// Mitsubishi GX Works2 project: vent_v02   PLC: FX3G
// Базовая структура управления вентиляциооной установкой

// global labels: Global1
VAR_GLOBAL
  xStart AT M10 : BOOL;  (* Переменная разрешения на работу установки *)
  xSeason AT M12 : BOOL;  (* Определение сезона 0 - Зима 1 - Лето *)
  xAlarm AT M1 : BOOL;  (* Общий статус Аварий 0 - нет 1 - Авария *)
  xWarning AT M2 : BOOL;  (* Общий статус предупреждений 0 - нет 1 - есть предупреждения *)
  dI_AlarmFreeze AT X000 : BOOL;  (* Авария термостата заморозки *)
  xAlarmSensors AT M7 : BOOL;  (* Общая аврия Датчиков - всне диапазона *)
  dI_AlarmPumpWater AT X001 : BOOL;  (* Авария насоса (сработка защиты) *)
  dI_AlarmMotorSupply AT X002 : BOOL;  (* Авария реле Вентилятора Притока *)
  dI_AlarmMotorExhaust AT X003 : BOOL;  (* Авария реле Вентилятора Вытяжки *)
  dI_WarnPresFilterSupply AT X007 : BOOL;  (* Авария пресостата фильтра Притока *)
  dI_WarnPresFilterExaust AT X006 : BOOL;  (* Авария пресостата фильтра Вытяжки *)
  dI_AlarmPresMotorSupply AT X004 : BOOL;  (* Авария пресостата вентилятора Притока *)
  dI_AlarmPresMotorExhaust AT X005 : BOOL;  (* Авария пресостата вентилятора Вытяжки *)
  xAlarmWarmWater AT M8 : BOOL;  (* Авария снижения температуры теплоносителя темплообменника - Требуется прогрев *)
  wDeltaTempOut AT D11 : INT;  (* Значение смещения показаний датчика (корректировка) *)
  wDeltaTempInRoom AT D10 : INT;  (* Значение смещения показаний датчика (корректировка) *)
  wDeltaTempFromRoom AT D9 : INT;  (* Значение смещения показаний датчика (корректировка) *)
  wDeltaTempEmpty AT D8 : INT;  (* Значение смещения показаний датчика (корректировка) *)
  xAlarmSensorOut AT M6 : BOOL;  (* Авария датчика Наружней температуры *)
  xAlarmSensorInRoom AT M5 : BOOL;  (* Авария датчика температуры Подачи В помещение *)
  xAlarmSensorFromRoom AT M4 : BOOL;  (* Авария датчика температуры забираемого ИЗ помещения *)
  xAlarmSensorEmpty AT M3 : BOOL;  (* Авария датчика температуры *)
  iR_TempOut AT D6 : WORD;  (* Значение сопротивление линии связи резистивного датчика *)
  iR_TempInRoom AT D5 : WORD;  (* Значение сопротивление линии связи резистивного датчика *)
  iR_TempFromRoom AT D4 : WORD;  (* Значение сопротивление линии связи резистивного датчика *)
  iRTempEmpty AT D7 : WORD;  (* Значение сопротивление линии связи резистивного датчика *)
  dO_PumpStart AT Y004 : BOOL;  (* Разрешение на работу Насоса контура водяного теплообменника *)
  dO_SupplyMotorStart AT Y003 : BOOL;  (* Разрешение на запуск Вентилятора Притока *)
  dO_ExhaustMotorStart AT Y001 : BOOL;  (* Разрешение на запуск Вентилятора Вытяжки *)
  dO_SupplyDamperStart AT Y002 : BOOL;  (* Разрешение на открытие Заслонки Притока *)
  dO_ExhaustDamperStart AT Y000 : BOOL;  (* Разрешение на открытие Заслонки Вытяжки *)
  iDelayStart AT D131 : WORD;  (* Значение задержки (общее) *)
  iDelaySupplyMotor AT D3 : WORD;  (* Значение задержки пуска Вентилятора Притока *)
  iDelayExhaustMotor AT D1 : WORD;  (* Значение задержки пуска Вентилятора Вытяжки *)
  iDelayDamper AT D132 : WORD;  (* Значение задержки открытия заслонки *)
  xUserStart AT M11 : BOOL;  (* Переменная изменяемая Пользователем для разрешения работы *)
  xUserSeason AT M13 : BOOL;  (* Переменная изменяемая Пользователем для выбора Сезона *)
  xUserArarmReset AT M14 : BOOL;  (* Переменная изменяемая Пользователем для сброса общего флага Аварий *)
  xAlarmCritical AT M0 : BOOL;  (* Cтатус критических Аварий 0 - нет 1 - Авария *)
  xInit AT M15 : BOOL;  (* Переменная разрешающая иницилизацию при старте *)
  aI_TempOut AT D14 : INT;  (* AI_0 Датчик наружней температуры D8030 *)
  aI_TempSupply AT D15 : INT;  (* AI_1 Датчик притока (температуры подачи в помещение)  D8031 *)
  aI_TempWater AT D16 : INT;  (* AI_2 Датчик обратной воды  D8032 *)
  aI_TempRecupOut AT D17 : INT;  (* AI_3 Датчик температуры за рекуператором  D8033 *)
  aO_1 AT D8050 : REAL;  (* AO_ Первый аналоговый D8050 *)
  aO_2 AT D8051 : REAL;  (* AO_ Второй аналоговый выход D8051 *)
  iUserTempSummer AT D128 : INT;  (* Температура перехода на летний режим *)
  iUserTemWinter AT D129 : INT;  (* Температура перехода на зимний режим *)
  aI_TempFromRoom AT D18 : INT;  (* AI_4 Датчик вытяжной температуры из помещения D8034 *)
  iUserAccess AT D40 : WORD;  (* Уровень доступа текущего пользователя *)
  iUserSetpointTempSupply AT D130 : INT;  (* Уставка заданная пользователем *)
  testTempOut AT D41 : INT;  (* Тестирование перехода   Зима/Лето *)
  iSetpointTempSupply AT D20 : INT;  (* Уставка температуры подачи Системная *)
  iUserSetpointTempWater AT D133 : INT;  (* Уставка контроля температуры теплоносителя (вода) *)
  iUserSetpointTempGlycol AT D134 : INT;  (* Уставка контроля температуры теплоносителя гликоль *)
  iUserSetpointTempAlarm AT D135 : INT;  (* Уставка контроля температуры Аварии *)
END_VAR

// task Task_01 (event TRUE, interval 0, priority 31): POU_01
// task Init (event M8002, interval 0, priority 24): Init
// task Process (event FALSE, interval T#150ms, priority 29): Process
// user libraries (not included): AlarmManger128v11, Utils

PROGRAM Init
VAR
  fbAmSet : AM_SET;
  fbAmInit : AM_INIT;
  fbAmIs : AM_HAS_ALARMS;
  fbAmBlockIs : AM_IS_BLOCK;
  fbAmEvents : AM_EVENT;
  fbAmRST : AM_RST;
  fbAmEventRST : AM_EVENT_RESET;
  inputType : BOOL;
END_VAR
(*Programm is run only one time when plc started to initiate alarms,  warnings and configuration settings *)


	AM_D_START :=3000; (* Start alarms library*)
	
	(* Critical Alarm signals*)
	 fbAmInit(iNum := 0, iSeverity :=3, iProcess :=1, xLock := TRUE,  xLatch := TRUE,  xBuzzer := TRUE ); (*Fire alarm *) 
	 
	  fbAmInit(iNum := 1, iSeverity :=2, iProcess :=2, xLock := TRUE,  xLatch := FALSE,  xBuzzer := TRUE ); (*Sensor alarm *) 


(* *)
END_PROGRAM

PROGRAM POU_01
VAR
  iStep : INT;
  fbAmSet : AM_SET;
  fbAmInit : AM_INIT;
  fbAmIs : AM_HAS_ALARMS;
  fbAmBlockIs : AM_IS_BLOCK;
  fbAmEvents : AM_EVENT;
  fbAmRST : AM_RST;
  fbAmEventRST : AM_EVENT_RESET;
  localSeasonTriger : BOOL;
  icountMin : INT;
  init : INT;
  currentTemp : INT;
  couner : INT;
END_VAR
(* RST( MEP( xManualWorks ) , xAutoWorks );
RST( MEP(xAutoWorks ) ,xManualWorks  );  *)
(* System can work only in one state Auto or Manual There is constol change*)
	
		fbAmIs(iProcessNum:= 2 ,iSeverity:= 2 ,Q:= xAlarmSensors);
		fbAmIs(iProcessNum:= 1, iSeverity:= 3 ,Q:= xAlarm );
 		IF xInit = 0 OR xAlarm THEN  iStep := 0 ; 
 		ELSE 
 			iStep := 10;
 		END_IF; (* Проверяем была ли выполнена инициализация xInit = 1 Ули была то переходим на шаг 10 если нет - на шаг 0 *)

fbAmRST(IN:= M10 );

CASE iStep OF
	0: (* Init  - Инициализация Задаем начальные значения переменным*)
	IF xInit = 0  THEN 
		dO_ExhaustDamperStart := 0;
		dO_SupplyDamperStart := 0;
		dO_ExhaustMotorStart := 0;
		dO_SupplyMotorStart := 0;
		xInit := 1;
	END_IF;

	
	10: (* Base *)
;
	20: (* Manage *)
;
	
	
	100: (* Alarm *)
		;
	END_CASE;
END_PROGRAM

PROGRAM Process
VAR
  fbAmSet : AM_SET;
END_VAR

fbAmSet(iNum:= 0, xState:= (NOT X000) ); (*Freeze Alarm*) 

fbAmSet(iNum:= 1 ,xState:= (D8030 = 4984) );
END_PROGRAM

FUNCTION SeasonControl
VAR_INPUT
  tempOut : INT;  (* Temp Outdore - Температура наружнего воздуха *)
  tempWinter : INT;  (* Temp for switch on Winter - Уставка перехода на Зимний режим *)
  tempSummer : INT;  (* Temp for switch on Summer - Уставка перехода на летний режим *)
  triger : BOOL;  (* 1 - was switch to winter 0 - was switch to summer *)
END_VAR
IF tempOut  <  tempWinter THEN 
		SeasonControl := 1; (* Output  Set flag - 1  to force switching to Winter *)
	ELSE 
		IF tempOut  > tempSummer THEN 
			SeasonControl := 0; (* Output  Set flag - 0  to force switching to Summer*)
		ELSE 
			SeasonControl := triger; (* Don't change r*)
		END_IF;

	END_IF;
END_FUNCTION

FUNCTION TestFunction
TestFunction := TRUE;
END_FUNCTION
